FUNCTION FC_Sum_int : INT
VAR_INPUT
	operand1 : INT;
	operand2 : INT;
END_VAR
VAR
END_VAR


FC_Sum_int := operand1 + operand2

END_FUNCTION

(* stored: Version 1.1.0.1
   POU FC_Sum_int: Id {7602be65-ed33-0c01-2310-e075aba6cb83}, SpecialFunc None *)
